SUBAPPLICATION Uebung_248_AX (* Wie Uebung_246_AX (Hoch/Runter auf 75/50/25%), zusaetzlich echter logiBUS_QDA_PWM-Ausgang Q1 zum Nachmessen *)
  (* Standard: 61499-2; Description: Copyright (c) 2026 Meisterschulen am Ostbahnhof This program and the accompanying materials are made available under the terms of the Eclipse Public License 2.0 which is available at https://www.eclipse.org/legal/epl-2.0/ SPDX-License-Identifier: EPL-2.0 *)
  (* Version 1.0, 2026-09-07, Franz Höpfinger, Meisterschulen am Ostbahnhof, initial API and implementation and/or initial documentation *)
  PACKAGE Uebungen;
  IMPORT logiBUS::io::DI::logiBUS_DI::Input_I1;
  IMPORT logiBUS::io::DI::logiBUS_DI::Input_I2;
  IMPORT Uebungen::const::UT::DefaultPool_Numeric::OutputNumber_N3_N;
  IMPORT logiBUS::io::DQ::logiBUS_DO::Output_Q1;
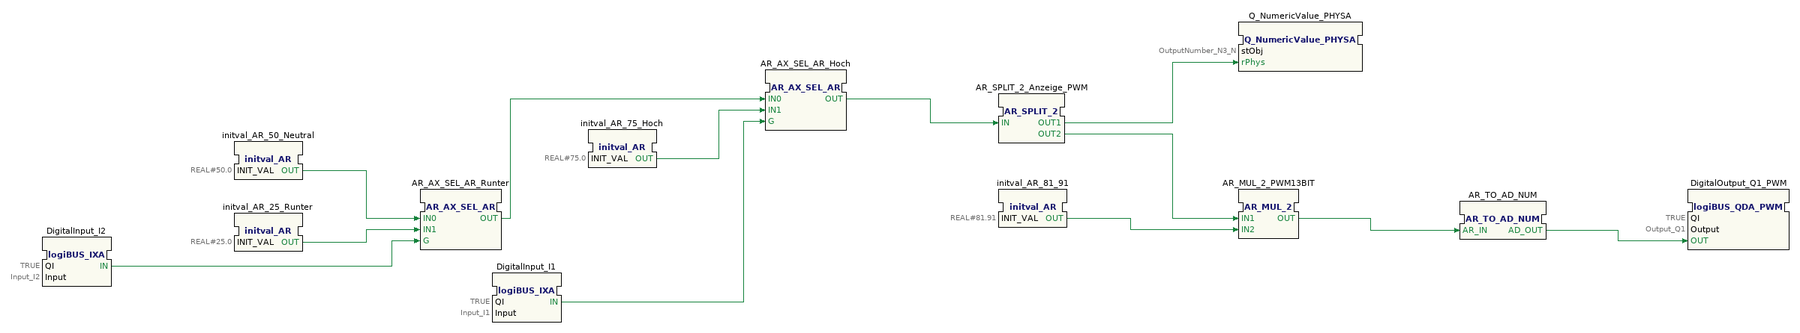
  (* 0-100% Tastgrad = 0-8191 (13-Bit LEDC, siehe RampLimitFS_TO_logiBUS_QDA_PWM_OPC.SUB in MyLib_AX-1.0.0): Faktor 81,91 = 8191/100. Mit Multimeter/Oszilloskop an Q1 gegen GND: Mittelwert = Tastgrad% x Versorgungsspannung - bei 25/50/75% Tastgrad direkt vergleichbar mit den PVEA-Sollspannungen 0,25/0,50/0,75 x U_DC. *)
  FBS
    DigitalInput_I1 : logiBUS::io::DI::logiBUS_IXA(QI := TRUE, Input := Input_I1);
    DigitalInput_I2 : logiBUS::io::DI::logiBUS_IXA(QI := TRUE, Input := Input_I2);
    initval_AR_50_Neutral : adapter::types::unidirectional::AR::initval::initval_AR(INIT_VAL := REAL#50.0);
    initval_AR_25_Runter : adapter::types::unidirectional::AR::initval::initval_AR(INIT_VAL := REAL#25.0);
    initval_AR_75_Hoch : adapter::types::unidirectional::AR::initval::initval_AR(INIT_VAL := REAL#75.0);
    AR_AX_SEL_AR_Runter : adapter::iec61131::selection::AR_AX_SEL_AR;
    AR_AX_SEL_AR_Hoch : adapter::iec61131::selection::AR_AX_SEL_AR;
    AR_SPLIT_2_Anzeige_PWM : adapter::events::unidirectional::AR_SPLIT_2;
    Q_NumericValue_PHYSA : isobus::UT::Q::Q_NumericValue_PHYSA(stObj := OutputNumber_N3_N);
    AR_MUL_2_PWM13BIT : adapter::iec61131::arithmetic::AR_MUL_2;
    initval_AR_81_91 : adapter::types::unidirectional::AR::initval::initval_AR(INIT_VAL := REAL#81.91);
    DigitalOutput_Q1_PWM : logiBUS::io::DQ::logiBUS_QDA_PWM(QI := TRUE, Output := Output_Q1);
    AR_TO_AD_NUM : adapter::conversion::unidirectional::AR_TO_AD_NUM;
  END_FBS
  ADAPTER_CONNECTIONS
    initval_AR_50_Neutral.OUT TO AR_AX_SEL_AR_Runter.IN0;
    initval_AR_25_Runter.OUT TO AR_AX_SEL_AR_Runter.IN1;
    DigitalInput_I2.IN TO AR_AX_SEL_AR_Runter.G;
    AR_AX_SEL_AR_Runter.OUT TO AR_AX_SEL_AR_Hoch.IN0;
    initval_AR_75_Hoch.OUT TO AR_AX_SEL_AR_Hoch.IN1;
    DigitalInput_I1.IN TO AR_AX_SEL_AR_Hoch.G;
    AR_AX_SEL_AR_Hoch.OUT TO AR_SPLIT_2_Anzeige_PWM.IN;
    AR_SPLIT_2_Anzeige_PWM.OUT1 TO Q_NumericValue_PHYSA.rPhys;
    AR_SPLIT_2_Anzeige_PWM.OUT2 TO AR_MUL_2_PWM13BIT.IN1;
    initval_AR_81_91.OUT TO AR_MUL_2_PWM13BIT.IN2;
    AR_MUL_2_PWM13BIT.OUT TO AR_TO_AD_NUM.AR_IN;
    AR_TO_AD_NUM.AD_OUT TO DigitalOutput_Q1_PWM.OUT;
  END_CONNECTIONS
END_SUBAPPLICATION
